// TIA Portal V20 export
TYPE "typeCmControlNode"
// stored: Namespace Unit1.Em0
   STRUCT
      interlock { ExternalWritable := 'False'} : "Unit1.Em0.typeCmControlNodeInterlock";
      brakeTest { S7_SetPoint := 'True'} : "Unit1.Em0.typeCmControlNodeBrakeTest";
   END_STRUCT;
END_TYPE
